(* PLC project Arduino Function Blocks, OpenPLC Arduino Function Blocks Library 1.0, author Thiago Alves *)
(* stored: creationDateTime 2021-11-11T02:33:11, modificationDateTime 2021-11-11T02:33:11 *)

(* Reads temperature from one DS18B20 one-wire sensor connected to the pin specified in PIN *)
FUNCTION_BLOCK DS18B20
  VAR_INPUT
    PIN : SINT;  (* Arduino pin where sensor is connected to *)
  END_VAR
  VAR_OUTPUT
    OUT : REAL;  (* Temperature output in Celsius *)
  END_VAR

            OUT := 0.0;
          
END_FUNCTION_BLOCK

(* Reads temperature from two DS18B20 one-wire sensors. Both sensors must be on the same bus connected to the pin specified in PIN *)
FUNCTION_BLOCK DS18B20_2_OUT
  VAR_INPUT
    PIN : SINT;  (* Arduino pin where sensor is connected to *)
  END_VAR
  VAR_OUTPUT
    OUT_0 : REAL;  (* Temperature output in Celsius *)
    OUT_1 : REAL;  (* Temperature output in Celsius *)
  END_VAR

            OUT := 0.0;
          
END_FUNCTION_BLOCK

(* Reads temperature from three DS18B20 one-wire sensors. All sensors must be on the same bus connected to the pin specified in PIN *)
FUNCTION_BLOCK DS18B20_3_OUT
  VAR_INPUT
    PIN : SINT;  (* Arduino pin where sensor is connected to *)
  END_VAR
  VAR_OUTPUT
    OUT_0 : REAL;  (* Temperature output in Celsius *)
    OUT_1 : REAL;  (* Temperature output in Celsius *)
    OUT_2 : REAL;  (* Temperature output in Celsius *)
  END_VAR

            OUT := 0.0;
          
END_FUNCTION_BLOCK

(* Reads temperature from four DS18B20 one-wire sensors. All sensors must be on the same bus connected to the pin specified in PIN *)
FUNCTION_BLOCK DS18B20_4_OUT
  VAR_INPUT
    PIN : SINT;  (* Arduino pin where sensor is connected to *)
  END_VAR
  VAR_OUTPUT
    OUT_0 : REAL;  (* Temperature output in Celsius *)
    OUT_1 : REAL;  (* Temperature output in Celsius *)
    OUT_2 : REAL;  (* Temperature output in Celsius *)
    OUT_3 : REAL;  (* Temperature output in Celsius *)
  END_VAR

            OUT := 0.0;
          
END_FUNCTION_BLOCK

(* Reads temperature from five DS18B20 one-wire sensors. All sensors must be on the same bus connected to the pin specified in PIN *)
FUNCTION_BLOCK DS18B20_5_OUT
  VAR_INPUT
    PIN : SINT;  (* Arduino pin where sensor is connected to *)
  END_VAR
  VAR_OUTPUT
    OUT_0 : REAL;  (* Temperature output in Celsius *)
    OUT_1 : REAL;  (* Temperature output in Celsius *)
    OUT_2 : REAL;  (* Temperature output in Celsius *)
    OUT_3 : REAL;  (* Temperature output in Celsius *)
    OUT_4 : REAL;  (* Temperature output in Celsius *)
  END_VAR

            OUT := 0.0;
          
END_FUNCTION_BLOCK

(* Add a BOOL variable to sync with the Arduino Cloud. VAR_NAME must have the same name as the variable set up in the Arduino IoT Cloud *)
FUNCTION_BLOCK CLOUD_ADD_BOOL
  VAR_INPUT
    VAR_NAME : STRING;
    BOOL_VAR : BOOL;
  END_VAR

            SSID := SSID;
          
END_FUNCTION_BLOCK

(* Add an DINT variable (Arduino int) to sync with the Arduino Cloud. VAR_NAME must have the same name as the variable set up in the Arduino IoT Cloud *)
FUNCTION_BLOCK CLOUD_ADD_DINT
  VAR_INPUT
    VAR_NAME : STRING;
    DINT_VAR : DINT;
  END_VAR

            SSID := SSID;
          
END_FUNCTION_BLOCK

(* Add a REAL variable (Arduino float) to sync with the Arduino Cloud. VAR_NAME must have the same name as the variable set up in the Arduino IoT Cloud *)
FUNCTION_BLOCK CLOUD_ADD_REAL
  VAR_INPUT
    VAR_NAME : STRING;
    REAL_VAR : REAL;
  END_VAR

            SSID := SSID;
          
END_FUNCTION_BLOCK

(* Setup and initialize Arduino Cloud communication. Must be called before adding any variables (properties). *)
FUNCTION_BLOCK CLOUD_BEGIN
  VAR_INPUT
    THING_ID : STRING;
    SSID : STRING;
    PASS : STRING;
  END_VAR

            SSID := SSID;
          
END_FUNCTION_BLOCK

(* Configures the CPU internal PWM peripheral to generate a PWM signal through hardware. If the CPU does not have a PWM peripheral, compiling this block will result in a compilation error. CHANNEL is the PWM channel number. For most Arduino boards that number is the pin number for the PWM capable pin. FREQ is the desired PWM frequency in Hz. DUTY is the PWM duty cycle (between 0 and 100). *)
FUNCTION_BLOCK PWM_CONTROLLER
  VAR_INPUT
    CHANNEL : SINT;  (* CHANNEL *)
    FREQ : REAL;  (* FREQ *)
    DUTY : REAL;  (* DUTY *)
  END_VAR
  VAR
    internal_ch : SINT;  (* internal_ch *)
    internal_freq : REAL;  (* internal_freq *)
    internal_duty : REAL;  (* internal_duty *)
  END_VAR
  VAR_OUTPUT
    SUCCESS : BOOL;  (* SUCCESS *)
  END_VAR

        
          IF CHANNEL < 1 THEN
            SUCCESS := FALSE;
            RETURN;
          END_IF;


          IF (CHANNEL <> internal_ch) OR (FREQ <> internal_freq) OR (DUTY <> internal_duty) THEN
            SUCCESS := TRUE;
          END_IF;

        
END_FUNCTION_BLOCK
